FUNCTION_BLOCK ABSTRACT Servo
VAR_INPUT CONSTANT
	bEnable : BOOL;
END_VAR
VAR_OUTPUT
	homeSet : BOOL;
	busy : BOOL;
	error : BOOL;
	
	position : REAL;
	targetPos : REAL;
END_VAR

END_FUNCTION_BLOCK

(* stored: Version 1.1.0.1, ProductVersion 3.1.4024.11
   POU Servo: Id {7c0cb4a8-1f86-45e8-a8fe-962ba57ecc76}, SpecialFunc None *)
